Fanuc KAREL source: KT00484.KL

PROGRAM KT00484
%NOLOCKGROUP
VAR
  P1: POSITION
  P2: XYZWPREXT
  OUT: POSITION
BEGIN
    P2.Y = 2.0
  OUT = P1 : P2
END KT00484
